(* IEC 61131-3 sources: UniTest/iecUnitTest_br/Library_tests/main, 2 files *)

(* ---- LocalVariables.var ---- *)
VAR
    testReporter : utTestReporter; (*Calculator for summaries of tests*)
END_VAR

(* ---- main.st ---- *)
PROGRAM _CYCLIC
    (*https://github.com/tkucic/iecUnitTest/blob/main/docs/docs/ns/Library_tests/prg/main.md*)
    testReporter(Results:=GVL.Results);
END_PROGRAM
